FUNCTION_BLOCK Merge4to1 (* Template for a Basic Function Block Type *)
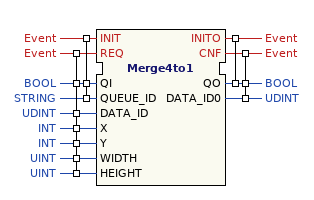
  EVENT_INPUT
    INIT WITH QI, QUEUE_ID; (* Initialization Request *)
    REQ WITH QI, DATA_ID, X, Y, WIDTH, HEIGHT; (* Normal Execution Request *)
  END_EVENT
  EVENT_OUTPUT
    INITO WITH QO; (* Initialization Confirm *)
    CNF WITH QO, DATA_ID0; (* Execution Confirmation *)
  END_EVENT
  VAR_INPUT
    QI : BOOL; (* Input event qualifier *)
    QUEUE_ID : STRING;
    DATA_ID : UDINT;
    X : INT;
    Y : INT;
    WIDTH : UINT;
    HEIGHT : UINT;
  END_VAR
  VAR_OUTPUT
    QO : BOOL; (* Output event qualifier *)
    DATA_ID0 : UDINT;
  END_VAR
END_FUNCTION_BLOCK
